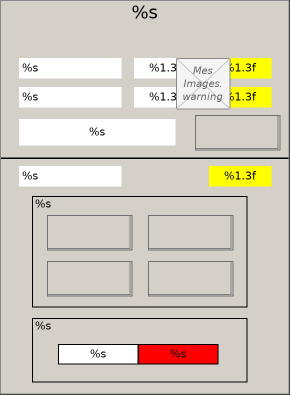
VISUALIZATION VISU_XTC  // 290x395
VAR_IN_OUT
	M_Input_Evap:		BLOCK_EVAP;
	M_Input_Ctrl:		BLOCK_XTC3;
	M_Input_QZ1:		BLOCK_XTAL6;
END_VAR
    GroupBox (0,144 290x251), invisible if: NOT M_Input_Ctrl.VISU_Show_Details
        Rectangle (0,14 290x237)
        RoundedRectangle (32,52 215x111), "%s", text list: 'TextList_IC6', text index: 4
        Button (47,71 85x35), input disabled if: NOT PRG_USER.ACTU_USER.MAINTENANCE OR NOT MACHINE.STATE_Manu, text list: 'TextList_IC6', text index: 5
            toggle M_Input_Ctrl.M_Start
        Button (47,117 85x35), input disabled if: NOT PRG_USER.ACTU_USER.MAINTENANCE OR NOT MACHINE.STATE_Manu, text list: 'TextList_IC6', text index: 6
            toggle M_Input_Ctrl.M_Stop
        Button (148,71 85x35), input disabled if: NOT PRG_USER.ACTU_USER.MAINTENANCE OR NOT MACHINE.STATE_Manu, text list: 'TextList_IC6', text index: 7
            toggle M_Input_Ctrl.M_RAZ_Thick
        Button (148,117 85x35), input disabled if: NOT PRG_USER.ACTU_USER.MAINTENANCE OR NOT MACHINE.STATE_Manu, text list: 'TextList_IC6', text index: 8
            toggle M_Input_Ctrl.M_Reset
        Textfield (19,22 102x20), "%s", text list: 'TextList_IC6', text index: 3
        Textfield (209,22 62x20), "%1.3f", text variable: M_Input_Ctrl.STATE_Power
        RoundedRectangle (32,174 215x64), "%s", text list: 'TextList_IC6', text index: 9
        Rectangle (58,200 80x20), "%s", text variable: M_Input_QZ1.MNEMO
        Rectangle (138,200 80x20), "OK", invisible if: M_Input_QZ1.STATE_NOK
        Rectangle (138,200 80x20), "%s", invisible if: NOT M_Input_QZ1.STATE_NOK, text list: 'TextList_IC6', text index: 10
    Rectangle (0,0 290x158), "%s", text variable: M_Input_Ctrl.MNEMO
    Textfield (19,58 102x20), "%s", text list: 'TextList_IC6', text index: 0
    Textfield (19,87 102x20), "%s", text list: 'TextList_IC6', text index: 1
    Textfield (209,58 62x20), "%1.3f", text variable: M_Input_Ctrl.STATE_Rate
    Textfield (209,87 62x20), "%1.3f", text variable: M_Input_Ctrl.STATE_Thickness
    Textfield (134,58 62x20), "%1.3f", text variable: M_Input_Evap.PRM_Rate, input disabled if: NOT Global_Variables.PRG_USER.ACTU_USER.MAINTENANCE OR NOT MACHINE.STATE_Manu
    Textfield (134,87 62x20), "%1.3f", text variable: M_Input_Evap.PRM_Thickness, input disabled if: NOT Global_Variables.PRG_USER.ACTU_USER.MAINTENANCE OR NOT MACHINE.STATE_Manu
    RoundedRectangle (19,119 156x26), "%s", text variable: M_Input_Ctrl.STATE_Phase
    Image (176,58 54x51), invisible if: NOT M_Input_Ctrl.STATE_NOK, image: MesImages.warning
    Button (195,115 85x35), text list: 'TextList_IC6', text index: 2
        toggle M_Input_Ctrl.VISU_Show_Details
END_VISUALIZATION

(* stored: Version 1.1.0.1, ProductVersion 3.1.4024.10
   Visu VISU_XTC: Id {ba92d797-9613-4742-b942-2171c40bc8bb} *)
